RoboDK station: roboticProjectFinal.rdk

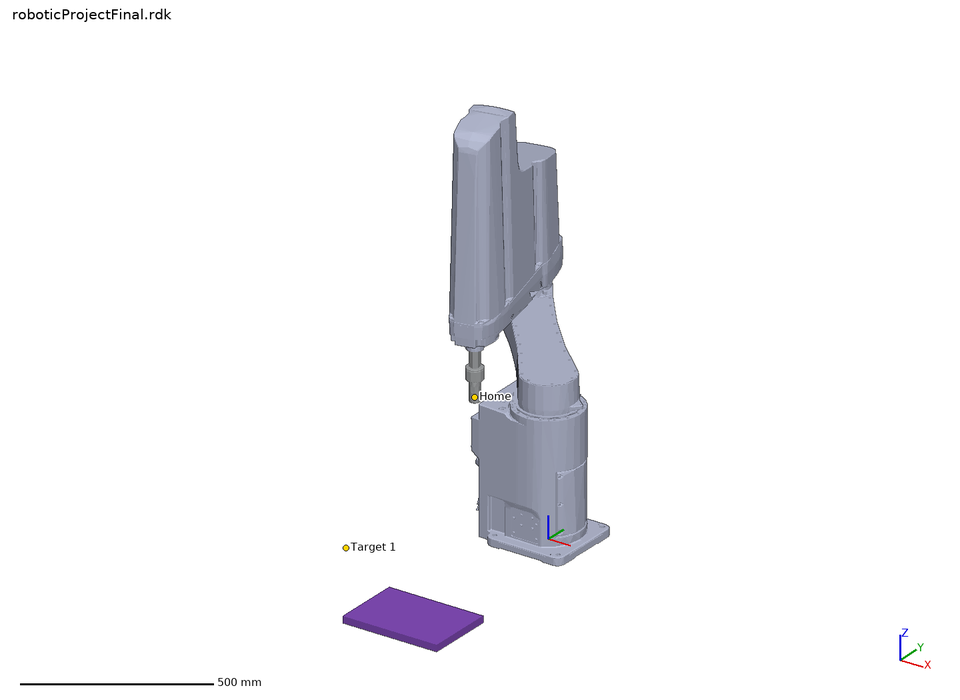
[picture v0: the station drawn from its stored meshes, robots at their saved joint values, targets as dots, program paths as lines]
Station roboticProjectFinal (saved by RoboDK 5.3.2). Poses are relative to the parent item; angles as X-Y-Z fixed-axis rotations.
  - frame Mitsubishi RH-20FRH8535 Base at (0, 0, 0) mm
    - robot Mitsubishi RH-20FRH8535: 4 axes, payload 20 kg, reach 850 mm, repeatability 0.025 mm
        modified DH rows (alpha deg, a mm, theta deg, d mm): 0, 0, 0, 0; 0, 525, 0, 0; 0, 325, 0, 0 linear; 180, 0, 0, 0
        joint limits [-132, -150, 0, -360] to [132, 150, 300, 360]; home [0, 0, 350, 0]; saved at [132, 150, 300, 0]
    - target Target 1 (joint target) at (-45.76, -848, 300) mm, rotated rx 0 ry 0 rz -90 deg; joints [-95, 5, 300, 0] of Mitsubishi RH-20FRH8535
    - target Home (joint target) at (-283.72, 72.25, 300) mm, rotated rx 0 ry 0 rz -78 deg; joints [132, 150, 300, 0] of Mitsubishi RH-20FRH8535
  - object Robotics Project A4 at (90, -740, 80) mm, rotated rx 0 ry 0 rz -90 deg, size 210 x 297 x 20 mm, geometry from Robotics Project A4.stl
  - Python program roboticsfinal11 (listed below)

--- Python program roboticsfinal11 ---
from robolink import *
from robodk import *
import json
RDK = Robolink()
robot = RDK.Item('', ITEM_TYPE_ROBOT)

scale = mbox('Enter the scale down value', entry=True)
scale = float(scale)
breakThreshold = mbox('Enter break away threshold value',entry=True)
breakThreshold= float(breakThreshold)

target= RDK.Item('Target 1')
home= RDK.Item('Home')

target_pose=target.Pose()

startPoint= target_pose.Pos()
robot.MoveJ(target)
with open('E:/Documents/Assignment Sem 1 4th Year/Robotics mini project/nameCoords.json') as data_file:
  dataCoords=json.load(data_file)
arrayNum = len(dataCoords)-1
for i in range(arrayNum):

  x= startPoint[0]+(dataCoords[i][0]/scale)
  y=startPoint[1]+(dataCoords[i][1]/scale)
  z= startPoint[2]-200

  breakPointX1=startPoint[0]+(dataCoords[i][0]/scale)
  breakPointX2=startPoint[0]+(dataCoords[i+1][0]/scale)

  breakPointY1=startPoint[1]+(dataCoords[i][1]/scale)
  breakPointY2=startPoint[1]+(dataCoords[i+1][1]/scale)

  breakDeltaX=breakPointX1-breakPointX2
  breakDeltaX = abs(breakDeltaX)

  breakDeltaY=breakPointY1-breakPointY2
  breakDeltaY = abs(breakDeltaY)

  if breakDeltaX > breakThreshold:
    z= startPoint[2]

  if breakDeltaY > breakThreshold:
    z= startPoint[2]


  target_pose.setPos([x,y,z])
  robot.MoveL(target_pose)
robot.MoveJ(target)
robot.RunInstruction('Program_Done')
